TYPE ST_Recipe :
	STRUCT
		Axis : ST_AxisRecipe;
	END_STRUCT
END_TYPE

(* stored: Version 1.1.0.1, ProductVersion 3.1.4026.18
   DUT ST_Recipe: Id {3b38cf75-e92b-4d0a-87b3-c5fc21ac940f} *)
